INTERFACE I_CalcLREAL EXTENDS I_Fallible


METHOD Calculate : LREAL
END_METHOD

END_INTERFACE

(* stored: Version 1.1.0.1
   Itf I_CalcLREAL: Id {5d461b0f-5eb0-46d4-89ed-d12b402454d0}
   Method Calculate: Id {01fcd5ca-c5aa-44a6-bbf6-7c6df2be8780} *)
